Staubli VAL3: GetArcLength.pgx

public program GetArcLength(trsf& x_trSource[], num& x_nLength, bool& x_bRes)
  local frame l_fFrame
  local trsf l_trCenter
  local num l_nDia
  local num l_nLength
  local num l_nAngle
  local trsf l_trBuff
begin
  //获得圆弧长度

  call Circumcircle(x_trSource,l_trCenter,l_nDia,x_bRes)
  if !x_bRes or l_nDia<=0
    x_bRes=false
    return
  endIf






  //计算三点的圆弧长度
  //2015.09.09
  //

  //强制二分，避免出现多边弧的问题
  l_trBuff=interpolateC(x_trSource[0],x_trSource[1],x_trSource[2],0.5)



  l_nLength=distance(x_trSource[0],l_trBuff)
  l_nAngle=asin(l_nLength/l_nDia)
  x_nLength=l_nAngle/180*l_nLength


  l_nLength=distance(l_trBuff,x_trSource[2])
  l_nAngle=asin(l_nLength/l_nDia)
  x_nLength=l_nAngle/180*l_nLength+x_nLength








end
